Yaskawa INFORM job: X2_51(P)(-165,-90).JBI

/JOB
//NAME X2_51(P)(-165,-90)
//POS
///NPOS 337,337,337,21,0,0
///TOOL 0
///POSTYPE PULSE
///PULSE
C00000=39612,-76551,-106625,-19964,71626,-76894
C00001=136747,-74177,-105509,-19364,71994,-77223
C00002=161484,-91945,-110261,-14957,103238,-71453
C00003=160103,-106044,-63154,-4849,72775,-63697
C00004=161344,-104617,-58318,-4903,70612,-63188
C00005=161861,-103966,-56335,-4926,69759,-62977
C00006=161974,-102590,-54020,-4947,69050,-62909
C00007=162012,-102745,-54357,-4943,69180,-62902
C00008=163250,-104574,-55005,-4953,68713,-62462
C00009=162012,-102745,-54357,-4943,69180,-62902
C00010=160245,-104918,-61242,-4863,72187,-63625
C00011=171505,-139740,-90933,-7250,74874,-61360
C00012=160934,-120333,-86405,-7656,81002,-65284
C00013=161678,-120105,-82177,-7691,78608,-64883
C00014=162014,-119639,-79976,-7711,77534,-64702
C00015=162103,-118683,-78296,-7724,77005,-64638
C00016=162142,-118788,-78603,-7719,77142,-64634
C00017=163383,-121045,-79330,-7709,76552,-64175
C00018=162142,-118788,-78603,-7719,77142,-64634
C00019=161077,-119352,-84635,-7663,80435,-65200
C00020=170862,-154578,-108681,-8518,79424,-59558
C00021=160995,-130363,-103106,-9103,87223,-63446
C00022=161741,-131140,-99278,-9095,84585,-62999
C00023=162088,-130949,-97067,-9096,83376,-62793
C00024=162168,-130176,-95642,-9101,82912,-62732
C00025=162238,-130240,-95916,-9096,83053,-62718
C00026=163482,-133028,-96761,-9062,82290,-62238
C00027=162238,-130240,-95916,-9096,83053,-62718
C00028=161170,-129514,-101410,-9099,86642,-63344
C00029=164342,-146461,-115997,5708,80531,-78436
C00030=172620,-131260,-102348,10866,75066,-76115
C00031=174663,-130573,-98097,10735,72570,-75614
C00032=175557,-129771,-95630,10687,71364,-75403
C00033=175655,-129031,-94295,10701,70918,-75408
C00034=175682,-129209,-94620,10692,71020,-75389
C00035=177260,-131621,-95369,10541,70050,-74910
C00036=175682,-129209,-94620,10692,71020,-75389
C00037=172786,-130448,-100678,10875,74444,-76112
C00038=185712,-152871,-107287,9933,65474,-72285
C00039=172557,-120691,-85253,11157,70075,-76596
C00040=174600,-119310,-80674,11059,67728,-76082
C00041=175498,-118200,-77996,11031,66549,-75868
C00042=175592,-117418,-76647,11054,66116,-75875
C00043=175604,-117590,-76985,11043,66232,-75860
C00044=177181,-119548,-77634,10892,65428,-75363
C00045=175604,-117590,-76985,11043,66232,-75860
C00046=172709,-119718,-83491,11178,69480,-76597
C00047=183041,-134830,-88553,10500,63578,-73433
C00048=171873,-105200,-60293,14264,60373,-76350
C00049=174332,-102742,-55136,14143,58110,-75711
C00050=175369,-101410,-52567,14107,57068,-75452
C00051=175489,-100273,-50681,14176,56489,-75483
C00052=175484,-100515,-51075,14158,56604,-75470
C00053=177059,-102096,-51658,13960,55908,-74954
C00054=175484,-100515,-51075,14158,56604,-75470
C00055=174474,-101588,-53199,14210,57504,-75737
C00056=172007,-104102,-58400,14326,59768,-76379
C00057=145534,-132844,-96218,416,74991,-72838
C00058=145515,-153724,-122450,337,32933,-72823
C00059=145515,-153724,-122450,337,32933,-72823
C00060=145977,-137385,-98995,123,44015,-76512
C00061=126650,-119622,-94060,17558,35096,-87270
C00062=146093,-91262,-32695,-9242,9662,-72789
C00063=160671,-30783,15668,-32982,16065,-44517
C00064=161338,-23358,24708,-37738,14871,-42214
C00065=161591,-20267,28531,-39994,14370,-41134
C00066=161710,-18499,31905,-43322,13534,-39587
C00067=161697,-18674,31599,-43019,13601,-39728
C00068=160818,-16173,33693,-41566,13229,-40545
C00069=161697,-18674,31599,-43019,13601,-39728
C00070=161443,-21835,27676,-40467,14093,-40942
C00071=160779,-29405,18429,-35142,15276,-43501
C00072=135154,-32069,12634,-42029,20998,-54645
C00073=134732,-25138,21651,-45349,19348,-53134
C00074=134570,-22247,25451,-46978,18672,-52394
C00075=134606,-20594,28698,-49618,17908,-51149
C00076=134580,-20854,28257,-49268,17988,-51317
C00077=134270,-18078,30511,-48869,17866,-51557
C00078=134580,-20854,28257,-49268,17988,-51317
C00079=135167,-30880,15161,-43750,20301,-53823
C00080=130526,-37728,8761,-34606,19495,-58724
C00081=121050,-28931,19594,-23215,15148,-65580
C00082=121021,-21638,29205,-26791,13167,-63944
C00083=121010,-18566,33292,-28698,12330,-63076
C00084=121003,-15436,36219,-29112,12158,-62888
C00085=120965,-16234,35448,-28882,12203,-63000
C00086=120957,-14841,38575,-31824,11150,-61665
C00087=120965,-16234,35448,-28882,12203,-63000
C00088=121002,-26728,21497,-23181,15100,-65604
C00089=121044,-28941,19424,-23061,15238,-65652
C00090=121016,-21660,29021,-26586,13257,-64038
C00091=121005,-18594,33102,-28462,12419,-63184
C00092=120998,-15466,36026,-28869,12247,-63000
C00093=120970,-16325,35175,-28625,12311,-63116
C00094=120961,-14943,38290,-31508,11257,-61807
C00095=120970,-16325,35175,-28625,12311,-63116
C00096=121007,-26794,21256,-23025,15206,-65675
C00097=146102,-87320,-26882,-11020,8134,-71987
C00098=145977,-137385,-98995,123,44015,-76512
C00099=112492,-157991,-119063,-2457,0,-76621
C00100=-11604,-169116,-125244,-11553,23484,-75880
C00101=-142186,-149365,-128787,911,0,-68169
C00102=-169394,-149435,-128797,930,71008,-68172
C00103=-146318,-131671,-100763,953,62874,-68185
C00104=-112829,-124197,-91749,2815,37541,-68231
C00105=-106317,-89557,-31431,-13456,10069,-57380
C00106=-82305,-48194,-2702,-1068,13384,-54980
C00107=-80735,-41443,4673,-5524,12373,-52723
C00108=-80143,-38689,7738,-7432,11949,-51767
C00109=-80007,-37233,10634,-8542,10936,-51243
C00110=-79998,-37162,10484,-8474,11064,-51273
C00111=-80961,-34830,12178,-5427,11144,-52800
C00112=-79998,-37162,10484,-8474,11064,-51273
C00113=-80428,-35938,10350,-6726,11733,-52131
C00114=-78778,-34690,11115,-11291,12069,-49811
C00115=-80428,-35938,10350,-6726,11733,-52131
C00116=-82562,-45500,-282,-411,13276,-55316
C00117=-92230,-47187,-3616,-43240,24199,-57639
C00118=-93096,-40890,4303,-45146,22607,-56839
C00119=-93429,-38304,7591,-46074,21957,-56442
C00120=-93338,-36887,10462,-48076,21279,-55468
C00121=-93324,-37096,10094,-47861,21367,-55569
C00122=-93984,-34586,11898,-46952,21176,-56108
C00123=-93324,-37096,10094,-47861,21367,-55569
C00124=-92116,-46106,-1290,-44710,23611,-56904
C00125=-91073,-53322,-8580,-41986,25230,-57812
C00126=-91939,-47488,-3032,-40883,24993,-58457
C00127=-92774,-41247,4932,-42701,23345,-57694
C00128=-93096,-38682,8241,-43585,22671,-57316
C00129=-93741,-35973,10491,-43009,22389,-57697
C00130=-93557,-36801,9788,-43160,22476,-57594
C00131=-93351,-35803,12350,-45165,21793,-56596
C00132=-93557,-36801,9788,-43160,22476,-57594
C00133=-92437,-45645,-1602,-40370,24830,-58783
C00134=-106116,-47899,-3414,-24973,19848,-68149
C00135=-106551,-41527,4610,-26418,18218,-67531
C00136=-106718,-38911,7943,-27146,17534,-67215
C00137=-107051,-36097,10252,-26581,17460,-67530
C00138=-106917,-36892,9642,-26842,17469,-67388
C00139=-106813,-35930,12180,-28635,16550,-66536
C00140=-106917,-36892,9642,-26842,17469,-67388
C00141=-106334,-45915,-1841,-24600,19835,-68356
C00142=-112836,-101934,-56773,3722,27473,-393
C00143=-146326,-133616,-103789,948,63737,26
C00144=-169394,-149435,-128797,930,71008,40
C00145=-130640,-113336,-116882,-25805,15754,2900
C00146=-135014,-119633,-103449,-15272,86576,5177
C00147=-145520,-105980,-62980,746,70150,73322
C00148=-146362,-104694,-58180,786,67864,73018
C00149=-146742,-103661,-55476,805,66734,72879
C00150=-146802,-102720,-53893,810,66245,72855
C00151=-146820,-102923,-54246,810,66358,72850
C00152=-147635,-104920,-54937,842,65765,72565
C00153=-146820,-102923,-54246,810,66358,72850
C00154=-145619,-104907,-61084,752,69535,73285
C00155=-171454,-106797,-63241,1567,70253,64421
C00156=-173073,-105087,-58310,1635,68130,63837
C00157=-173822,-103661,-55199,1669,66963,63564
C00158=-173907,-102906,-53963,1677,66592,63529
C00159=-173899,-103121,-54319,1675,66700,63533
C00160=-175454,-104758,-54906,1725,66251,62992
C00161=-173899,-103121,-54319,1675,66700,63533
C00162=-171598,-105684,-61333,1577,69654,64364
C00163=-171851,-142113,-91727,1629,69899,64268
C00164=-158429,-121713,-86926,1143,76935,68953
C00165=-159677,-121086,-82564,1192,74590,68504
C00166=-160262,-120091,-79675,1217,73333,68291
C00167=-160325,-119479,-78625,1221,73002,68266
C00168=-160351,-119548,-78930,1221,73155,68259
C00169=-161558,-121835,-79657,1263,72445,67838
C00170=-160351,-119548,-78930,1221,73155,68259
C00171=-158575,-120647,-85141,1149,76386,68898
C00172=-146231,-120412,-85894,9154,79904,67922
C00173=-146532,-120200,-81655,9220,77469,67638
C00174=-146707,-119317,-78712,9263,76149,67479
C00175=-146746,-118772,-77764,9274,75853,67443
C00176=-146790,-118881,-78072,9269,75989,67438
C00177=-147605,-121338,-78846,9287,75305,67107
C00178=-146790,-118881,-78072,9269,75989,67438
C00179=-146355,-119421,-84118,9167,79342,67838
C00180=-155393,-157537,-108482,12071,78573,60028
C00181=-146205,-130572,-102237,12226,86761,64000
C00182=-146506,-131303,-98376,12244,84115,63635
C00183=-146668,-130963,-95920,12261,82832,63453
C00184=-146721,-130297,-94717,12268,82450,63397
C00185=-146765,-130382,-95017,12263,82595,63396
C00186=-147581,-133401,-95913,12252,81739,63030
C00187=-146765,-130382,-95017,12263,82595,63396
C00188=-146330,-129706,-100552,12225,86202,63901
C00189=-158435,-132386,-103934,1126,81916,68996
C00190=-159685,-132645,-99938,1172,79342,68546
C00191=-160276,-131966,-97169,1195,77996,68332
C00192=-160335,-131435,-96228,1198,77691,68309
C00193=-160363,-131651,-96568,1198,77790,68300
C00194=-161574,-134495,-97414,1239,76868,67878
C00195=-160363,-131651,-96568,1198,77790,68300
C00196=-158581,-131628,-102288,1132,81296,68941
C00197=-156763,-87672,-103760,774,105674,87516
C00198=-169394,-149435,-128797,930,71008,83169
C00199=-150414,-86289,-54081,-474,90119,72869
C00200=-151266,-87748,-50943,-622,87433,72599
C00201=-152488,-87428,-48859,-834,86309,72204
C00202=-148147,-89589,-49139,4425,86731,74395
C00203=-146818,-89870,-51113,4706,87732,74872
C00204=-146666,-88304,-54215,4739,90428,75023
C00205=-138939,-90669,-55596,-9574,86239,77137
C00206=-140404,-91758,-52256,-9806,83488,76860
C00207=-142815,-91310,-50219,-10159,82191,76162
C00208=-154710,-86462,-48344,-11637,81955,72207
C00209=-152664,-87123,-50558,-11375,83242,72777
C00210=-150783,-86165,-53887,-11117,85991,73164
C00211=-154131,-121950,-82387,-8712,85987,67425
C00212=-148025,-100109,-75076,-5665,93909,72754
C00213=-148831,-100312,-70826,-5762,91146,72606
C00214=-146468,-101528,-70218,-8213,89409,73952
C00215=-156895,-95901,-68057,-9567,89811,70382
C00216=-156895,-97491,-71326,-9574,90990,70292
C00217=-153017,-102427,-75547,-11357,90518,71992
C00218=-151529,-98458,-73502,4508,98276,66494
C00219=-151321,-97538,-69606,4526,96344,66497
C00220=-152185,-98274,-68237,4332,95173,66163
C00221=-146393,-100560,-68313,8882,94911,67867
C00222=-146800,-100443,-69693,10119,95679,69043
C00223=-151558,-100768,-73356,9121,98301,67607
C00224=-156292,-129361,-96058,9643,101176,59304
C00225=-152402,-99580,-86113,11137,109464,61436
C00226=-153129,-103579,-84123,10707,106340,60878
C00227=-153762,-104985,-82590,10439,104784,60514
C00228=-145239,-109230,-83490,14196,102512,63288
C00229=-141027,-109993,-86316,13674,102607,64868
C00230=-140829,-106100,-88459,13958,105801,65311
C00231=-138968,-107947,-91550,-9748,99253,76121
C00232=-140436,-111637,-89327,-9854,95856,75879
C00233=-143265,-112181,-87516,-10198,94133,75040
C00234=-154691,-105452,-85498,-11618,94761,71024
C00235=-152715,-105048,-87091,-11430,96209,71575
C00236=-150832,-103395,-97227,-11518,103428,71561
C00237=-124659,-112995,-107713,-28856,68615,65766
C00238=-126218,-114256,-117174,-36511,17097,46518
C00239=-148561,-148351,-134746,-2636,59820,4885
C00240=-157191,-155093,-133027,-2423,70817,-63833
C00241=-146254,-116377,-77147,999,56200,-68180
C00242=-107275,-71407,-14739,-39799,20998,-48318
C00243=-107236,-64792,-7336,-41859,20126,-47330
C00244=-107209,-61980,-4011,-43007,19687,-46782
C00245=-70112,-45989,3773,-54150,40066,-34286
C00246=-69774,-48485,443,-53474,40707,-34620
C00247=-68604,-54637,-7231,-52245,42284,-35133
C00248=-92320,-90311,-38101,-17507,21359,-69759
C00249=-104434,-95533,-39177,3441,13241,-85394
C00250=-104568,-88850,-32673,3945,12680,-85644
C00251=-104520,-86387,-29909,3952,12244,-85640
C00252=-67588,-70566,-24092,-47976,27768,-56046
C00253=-72044,-71463,-22366,-44090,19939,-45466
C00254=-72907,-74424,-25211,-42700,19719,-46246
C00255=-73002,-81137,-31884,-41377,20172,-46887
C00256=-111917,-134748,-95138,2307,25782,-38985
C00257=-112830,-118606,-82850,2996,34941,-68234
C00258=-146284,-125214,-92772,982,57715,-68183
C00259=-169394,-149435,-128797,930,71008,-68172
C00260=-133816,-149354,-128786,835,13880,-68173
C00261=-90671,-157974,-126979,-5410,0,-71957
C00262=-11604,-169116,-125244,-11553,23484,-75880
C00263=137287,-84892,-120500,-10191,64594,-76446
C00264=160620,-101266,-113002,-23179,68693,-67515
C00265=177556,-94372,-53425,-385,88988,-62741
C00266=179326,-95097,-49878,3,86437,-62164
C00267=179814,-95288,-47635,109,84959,-62011
C00268=167774,-103484,-50203,-2536,82158,-65798
C00269=167400,-103593,-52544,-2612,83531,-65942
C00270=166065,-103008,-56268,-2894,86078,-66424
C00271=166312,-127479,-80936,-5864,94766,-53062
C00272=158392,-93304,-69893,-8747,104686,-56339
C00273=159554,-95674,-67229,-8288,101981,-55739
C00274=159445,-96667,-65849,-8272,100624,-55685
C00275=147725,-102887,-67985,-11495,97353,-59463
C00276=147678,-102382,-69650,-11553,98605,-59595
C00277=146987,-100069,-72442,-11867,101354,-60101
C00278=154304,-136297,-99225,-6964,97533,-61473
C00279=152227,-100568,-87835,-8146,108504,-62877
C00280=153116,-104646,-85864,-7761,105315,-62341
C00281=159148,-124823,-92360,-9877,92486,-59205
C00282=144137,-132852,-94532,-12005,87729,-63907
C00283=143944,-126885,-94638,-11486,92524,-64465
C00284=145540,-135687,-103511,-12475,90096,-63617
C00285=148082,-100818,-99733,10674,107205,-74531
C00286=152803,-93035,-83606,23107,96838,-80328
C00287=154879,-96218,-81430,23079,93509,-80208
C00288=162734,-110375,-86778,19923,82294,-79319
C00289=172936,-99666,-82887,19315,82782,-75563
C00290=164774,-87312,-77814,23533,92874,-76681
C00291=167890,-98830,-87724,19097,86606,-76775
C00292=158633,-112297,-90822,23483,90242,-79469
C00293=153117,-105481,-75293,18446,87539,-80566
C00294=154070,-103992,-71187,18555,85650,-80517
C00295=161541,-113229,-74370,16909,77144,-78922
C00296=171872,-105466,-71629,16874,77244,-75258
C00297=165515,-96039,-68345,19422,85228,-76531
C00298=163213,-94486,-71315,19256,88254,-76871
C00299=168945,-117983,-78283,23930,79136,-80745
C00300=162859,-103904,-55417,26052,71934,-81289
C00301=166467,-103150,-51264,26590,68911,-80665
C00302=174261,-106144,-51758,25332,63333,-78665
C00303=185047,-97716,-49331,24449,62895,-74631
C00304=178605,-94860,-48677,26497,67666,-76392
C00305=170055,-106805,-62873,25975,72582,-78466
C00306=152982,-88821,-92221,4904,67346,-32106
C00307=145515,-153724,-122450,337,32933,46
C00308=145515,-153724,-122450,337,32933,46
C00309=145977,-137385,-98995,123,44015,44
C00310=84186,-58858,-9027,66870,52124,39353
C00311=87105,-53815,-2337,68349,49752,38990
C00312=88013,-52041,490,69129,48884,38670
C00313=128614,-57932,-1955,73297,23821,44535
C00314=127846,-60584,-5316,71867,24516,45096
C00315=125900,-66978,-12435,69921,26079,45715
C00316=123713,-86623,-29625,34014,27338,1409
C00317=121149,-57675,-2785,-2636,26737,-48399
C00318=121132,-57328,-2241,-2634,26580,-48403
C00319=121104,-54911,-3160,-2183,31831,-48629
C00320=158495,-44767,2170,-23903,39526,-29988
C00321=121132,-57338,-2123,-2642,26502,-48399
C00322=121149,-57624,-2567,-2646,26629,-48394
C00323=145977,-137385,-98995,123,44015,44
C00324=141323,-155575,-119470,2858,47354,-2051
C00325=136193,-54528,-31246,1392,38939,57192
C00326=133673,-4879,12102,671,34805,86301
C00327=129645,-10071,18191,6510,19037,82612
C00328=146465,2091,28934,7064,17500,85725
C00329=143182,-12622,11657,11660,20903,83241
C00330=129180,-33068,-6989,1774,26259,77639
C00331=129999,-18466,14492,894,20530,78149
C00332=103012,-15842,16412,36484,27005,57754
C00333=109108,-49067,-22735,24370,30989,64550
C00334=115971,-133718,-81561,22438,22383,66198
C00335=115971,-174253,-123740,18555,27203,68106
C00336=39612,-76551,-106625,-19964,71626,-76894
BC00000=295309,515546,1075139
BC00001=353519,294132,1075139
BC00002=353519,214242,1075139
BC00003=331202,150916,1075139
BC00004=331202,150916,1075139
BC00005=331202,150916,1075139
BC00006=331202,150916,1075139
BC00007=331202,150916,1075139
BC00008=331202,150916,1075139
BC00009=331202,150916,1075139
BC00010=331202,150916,1075139
BC00011=324436,118777,1075139
BC00012=324436,118777,1075139
BC00013=324436,118777,1075139
BC00014=324436,118777,1075139
BC00015=324436,118777,1075139
BC00016=324436,118777,1075139
BC00017=324436,118777,1075139
BC00018=324436,118777,1075139
BC00019=324436,118777,1075139
BC00020=321391,89351,1075139
BC00021=321391,89351,1075139
BC00022=321391,89351,1075139
BC00023=321391,89351,1075139
BC00024=321391,89351,1075139
BC00025=321391,89351,1075139
BC00026=321391,89351,1075139
BC00027=321391,89351,1075139
BC00028=321391,89351,1075139
BC00029=308521,79020,1075139
BC00030=308521,79020,1075139
BC00031=308521,79020,1075139
BC00032=308521,79020,1075139
BC00033=308521,79020,1075139
BC00034=308521,79020,1075139
BC00035=308521,79020,1075139
BC00036=308521,79020,1075139
BC00037=308521,79020,1075139
BC00038=308521,79020,1075139
BC00039=308654,108079,1075139
BC00040=308654,108079,1075139
BC00041=308654,108079,1075139
BC00042=308654,108079,1075139
BC00043=308654,108079,1075139
BC00044=308654,108079,1075139
BC00045=308654,108079,1075139
BC00046=308654,108079,1075139
BC00047=308654,108079,1075139
BC00048=315387,142542,1075139
BC00049=315387,142542,1075139
BC00050=315387,142542,1075139
BC00051=315387,142542,1075139
BC00052=315387,142542,1075139
BC00053=315387,142542,1075139
BC00054=315387,142542,1075139
BC00055=315387,142542,1075139
BC00056=315387,142542,1075139
BC00057=334019,183746,1075139
BC00058=334019,229146,1075139
BC00059=369517,393170,1075139
BC00060=369517,393170,1075139
BC00061=309272,310148,725948
BC00062=299317,286166,1016538
BC00063=320949,304869,1075139
BC00064=320949,304869,1075139
BC00065=320949,304869,1075139
BC00066=320949,304869,1075139
BC00067=320949,304869,1075139
BC00068=320949,304869,1075139
BC00069=320949,304869,1075139
BC00070=320949,304869,1075139
BC00071=320949,304869,1075139
BC00072=287778,324241,1075139
BC00073=287778,324241,1075139
BC00074=287778,324241,1075139
BC00075=287778,324241,1075139
BC00076=287778,324241,1075139
BC00077=287778,324241,1075139
BC00078=287778,324241,1075139
BC00079=287778,324241,1075139
BC00080=279976,328662,1075139
BC00081=264373,337505,1075139
BC00082=264373,337505,1075139
BC00083=264373,337505,1075139
BC00084=264373,337505,1075139
BC00085=264373,337505,1075139
BC00086=264373,337505,1075139
BC00087=264373,337505,1075139
BC00088=264373,337505,1075139
BC00089=317151,337442,1075139
BC00090=317151,337442,1075139
BC00091=317151,337442,1075139
BC00092=317151,337442,1075139
BC00093=317151,337442,1075139
BC00094=317151,337442,1075139
BC00095=317151,337442,1075139
BC00096=317151,337442,1075139
BC00097=324891,309494,1043787
BC00098=369517,393170,1075139
BC00099=372480,297840,1075139
BC00100=335939,159824,1075139
BC00101=387142,-83097,1073718
BC00102=387142,-83097,1073718
BC00103=354260,-55239,919482
BC00104=302473,-54215,830727
BC00105=299756,-34503,1018031
BC00106=266432,-33337,1015863
BC00107=266432,-33337,1015863
BC00108=266432,-33337,1015863
BC00109=266432,-33337,1015863
BC00110=266432,-33337,1015863
BC00111=266432,-33337,1015863
BC00112=266432,-33337,1015863
BC00113=266432,-33337,1015863
BC00114=266432,-33337,1015863
BC00115=266432,-33337,1015863
BC00116=266432,-33337,1015863
BC00117=284169,-51063,1035355
BC00118=284169,-51063,1035355
BC00119=284169,-51063,1035355
BC00120=284169,-51063,1035355
BC00121=284169,-51063,1035355
BC00122=284169,-51063,1035355
BC00123=284169,-51063,1035355
BC00124=284169,-51063,1035355
BC00125=283205,-57233,1023653
BC00126=282402,-62375,1013902
BC00127=282402,-62375,1013902
BC00128=282402,-62375,1013902
BC00129=282402,-62375,1013902
BC00130=282402,-62375,1013902
BC00131=282402,-62375,1013902
BC00132=282402,-62375,1013902
BC00133=282402,-62375,1013902
BC00134=251376,-67725,1013804
BC00135=251376,-67725,1013804
BC00136=251376,-67725,1013804
BC00137=251376,-67725,1013804
BC00138=251376,-67725,1013804
BC00139=251376,-67725,1013804
BC00140=251376,-67725,1013804
BC00141=251376,-67725,1013804
BC00142=302473,-54215,999708
BC00143=354260,-55239,903923
BC00144=387142,-83097,1073718
BC00145=343892,52052,1075139
BC00146=340737,74809,1075139
BC00147=324434,99527,1075139
BC00148=324434,99527,1075139
BC00149=324434,99527,1075139
BC00150=324434,99527,1075139
BC00151=324434,99527,1075139
BC00152=324434,99527,1075139
BC00153=324434,99527,1075139
BC00154=324434,99527,1075139
BC00155=316013,112625,1075139
BC00156=316013,112625,1075139
BC00157=316013,112625,1075139
BC00158=316013,112625,1075139
BC00159=316013,112625,1075139
BC00160=316013,112625,1075139
BC00161=316013,112625,1075139
BC00162=316013,112625,1075139
BC00163=304877,137904,1075139
BC00164=304877,137904,1075139
BC00165=304877,137904,1075139
BC00166=304877,137904,1075139
BC00167=304877,137904,1075139
BC00168=304877,137904,1075139
BC00169=304877,137904,1075139
BC00170=304877,137904,1075139
BC00171=304877,137904,1075139
BC00172=308833,132707,1075139
BC00173=308833,132707,1075139
BC00174=308833,132707,1075139
BC00175=308833,132707,1075139
BC00176=308833,132707,1075139
BC00177=308833,132707,1075139
BC00178=308833,132707,1075139
BC00179=308833,132707,1075139
BC00180=303080,163439,1075139
BC00181=303080,163439,1075139
BC00182=303080,163439,1075139
BC00183=303080,163439,1075139
BC00184=303080,163439,1075139
BC00185=303080,163439,1075139
BC00186=303080,163439,1075139
BC00187=303080,163439,1075139
BC00188=303080,163439,1075139
BC00189=304913,167110,1075139
BC00190=304913,167110,1075139
BC00191=304913,167110,1075139
BC00192=304913,167110,1075139
BC00193=304913,167110,1075139
BC00194=304913,167110,1075139
BC00195=304913,167110,1075139
BC00196=304913,167110,1075139
BC00197=340038,100851,1073718
BC00198=340038,100851,1073718
BC00199=318440,111564,1057595
BC00200=318440,111564,1057595
BC00201=318440,111564,1057593
BC00202=318440,111564,1057595
BC00203=318440,111564,1057595
BC00204=318440,111564,1057595
BC00205=310795,111718,1057781
BC00206=310795,111718,1057781
BC00207=310795,111718,1057781
BC00208=310795,111718,1057781
BC00209=310795,111718,1057781
BC00210=310795,111718,1057781
BC00211=314493,146927,1075139
BC00212=311302,144606,1075139
BC00213=311302,144606,1075139
BC00214=311090,144452,1075139
BC00215=311090,144452,1075139
BC00216=311090,144452,1075139
BC00217=310912,144322,1075139
BC00218=309663,144665,1075139
BC00219=309663,144665,1075139
BC00220=309663,144665,1075139
BC00221=309663,144665,1075139
BC00222=309663,144665,1075139
BC00223=309663,144665,1075139
BC00224=293187,178635,1075139
BC00225=300015,175953,1075139
BC00226=300015,175953,1075139
BC00227=300015,175953,1075139
BC00228=300015,175953,1075139
BC00229=300015,175953,1075139
BC00230=300015,175953,1075139
BC00231=311011,173433,1075139
BC00232=311011,173433,1075139
BC00233=311011,173433,1075139
BC00234=311011,173433,1075139
BC00235=311011,173433,1075139
BC00236=311011,173433,1075139
BC00237=311721,119711,1075139
BC00238=312616,52052,1075139
BC00239=363630,-40460,1074166
BC00240=387142,-83097,1073718
BC00241=354260,-55239,1037445
BC00242=264595,-32771,1007498
BC00243=264595,-32771,1007498
BC00244=264595,-32771,1007498
BC00245=264595,-32771,1007498
BC00246=264595,-32771,1007498
BC00247=264595,-32771,1007498
BC00248=281388,-13085,953726
BC00249=292015,-7655,938135
BC00250=292015,-7655,938135
BC00251=292015,-7655,938135
BC00252=292015,-7655,938135
BC00253=292015,-7655,938135
BC00254=292015,-7655,938135
BC00255=292015,-7655,938135
BC00256=305209,-34503,728557
BC00257=302473,-54215,875335
BC00258=354260,-55239,995141
BC00259=387142,-83097,1073718
BC00260=387142,-83097,1073718
BC00261=392686,38993,1074432
BC00262=335939,159824,1075139
BC00263=353801,266119,1075139
BC00264=381880,223521,1075139
BC00265=325796,119524,1075139
BC00266=325796,119524,1075139
BC00267=325796,119524,1075139
BC00268=325796,119524,1075139
BC00269=325796,119524,1075139
BC00270=325796,119524,1075139
BC00271=298605,97380,1075139
BC00272=306786,105313,1075139
BC00273=306786,105313,1075139
BC00274=306786,105313,1075139
BC00275=306786,105313,1075139
BC00276=306786,105313,1075139
BC00277=306786,105313,1075139
BC00278=296424,73357,1075139
BC00279=304436,81384,1075139
BC00280=304436,81384,1075139
BC00281=304436,81384,1075139
BC00282=304436,81384,1075139
BC00283=304436,81384,1075139
BC00284=304436,81384,1075139
BC00285=314150,82141,1075139
BC00286=318449,85788,1075139
BC00287=318449,85788,1075139
BC00288=318449,85788,1075139
BC00289=318449,85788,1075139
BC00290=318449,85788,1075139
BC00291=318449,85788,1075139
BC00292=319675,83840,1075139
BC00293=303619,103646,1075139
BC00294=303619,103646,1075139
BC00295=303619,103646,1075139
BC00296=303619,103646,1075139
BC00297=303619,103646,1075139
BC00298=303619,103646,1075139
BC00299=318801,93459,1075139
BC00300=319660,117178,1064998
BC00301=319660,117178,1064998
BC00302=319660,117178,1064998
BC00303=319660,117178,1064998
BC00304=319660,117178,1064998
BC00305=319660,117178,1064998
BC00306=339598,204159,1070920
BC00307=334019,229146,1075139
BC00308=369517,393170,1075139
BC00309=369517,393170,1075139
BC00310=279240,278181,995341
BC00311=279240,278181,995341
BC00312=279240,278181,995341
BC00313=279240,278181,995341
BC00314=279240,278181,995341
BC00315=279240,278181,995341
BC00316=306644,283045,1033505
BC00317=336539,288351,1075139
BC00318=333822,285094,1054529
BC00319=332736,283791,1045508
BC00320=332727,283791,1045508
BC00321=279880,285191,1054163
BC00322=282597,288448,1075139
BC00323=369517,393170,1075139
BC00324=209346,479306,1075139
BC00325=169680,397657,995179
BC00326=150190,357539,955892
BC00327=150190,357539,955892
BC00328=150190,357539,955892
BC00329=150190,357539,955892
BC00330=150190,357539,955892
BC00331=150190,357539,955892
BC00332=150190,357539,955892
BC00333=150190,357539,955892
BC00334=150190,357539,955892
BC00335=150190,552519,961001
BC00336=295309,515546,1075139
EC00000=1463287,372643
EC00001=1463287,372643
EC00002=1463287,372643
EC00003=1463287,372643
EC00004=1463287,372643
EC00005=1463287,372643
EC00006=1463287,372643
EC00007=1463287,372643
EC00008=1463287,372643
EC00009=1463287,372643
EC00010=1463287,372643
EC00011=1463287,372643
EC00012=1463287,372643
EC00013=1463287,372643
EC00014=1463287,372643
EC00015=1463287,372643
EC00016=1463287,372643
EC00017=1463287,372643
EC00018=1463287,372643
EC00019=1463287,372643
EC00020=1463287,372643
EC00021=1463287,372643
EC00022=1463287,372643
EC00023=1463287,372643
EC00024=1463287,372643
EC00025=1463287,372643
EC00026=1463287,372643
EC00027=1463287,372643
EC00028=1463287,372643
EC00029=1463287,372643
EC00030=1463287,372643
EC00031=1463287,372643
EC00032=1463287,372643
EC00033=1463287,372643
EC00034=1463287,372643
EC00035=1463287,372643
EC00036=1463287,372643
EC00037=1463287,372643
EC00038=1463287,372643
EC00039=1463287,372643
EC00040=1463287,372643
EC00041=1463287,372643
EC00042=1463287,372643
EC00043=1463287,372643
EC00044=1463287,372643
EC00045=1463287,372643
EC00046=1463287,372643
EC00047=1463287,372643
EC00048=1463287,372643
EC00049=1463287,372643
EC00050=1463287,372643
EC00051=1463287,372643
EC00052=1463287,372643
EC00053=1463287,372643
EC00054=1463287,372643
EC00055=1463287,372643
EC00056=1463287,372643
EC00057=1463287,372643
EC00058=1463287,372643
EC00059=1463287,372643
EC00060=1463287,372643
EC00061=1463287,372643
EC00062=1463287,372643
EC00063=1463287,372643
EC00064=1463287,372643
EC00065=1463287,372643
EC00066=1463287,372643
EC00067=1463287,372643
EC00068=1463287,372643
EC00069=1463287,372643
EC00070=1463287,372643
EC00071=1463287,372643
EC00072=1463287,372643
EC00073=1463287,372643
EC00074=1463287,372643
EC00075=1463287,372643
EC00076=1463287,372643
EC00077=1463287,372643
EC00078=1463287,372643
EC00079=1463287,372643
EC00080=1463287,372643
EC00081=1463287,372643
EC00082=1463287,372643
EC00083=1463287,372643
EC00084=1463287,372643
EC00085=1463287,372643
EC00086=1463287,372643
EC00087=1463287,372643
EC00088=1463287,372643
EC00089=1463287,372643
EC00090=1463287,372643
EC00091=1463287,372643
EC00092=1463287,372643
EC00093=1463287,372643
EC00094=1463287,372643
EC00095=1463287,372643
EC00096=1463287,372643
EC00097=1463287,372643
EC00098=1463287,372643
EC00099=1463287,372643
EC00100=1595090,-179995
EC00101=1729339,-740307
EC00102=1729339,-740307
EC00103=1729339,-740307
EC00104=1729339,-740307
EC00105=1729339,-740307
EC00106=1729339,-740307
EC00107=1729339,-740307
EC00108=1729339,-740307
EC00109=1729339,-740307
EC00110=1729339,-740307
EC00111=1729339,-740307
EC00112=1729339,-740307
EC00113=1729339,-740307
EC00114=1729339,-740307
EC00115=1729339,-740307
EC00116=1729339,-740307
EC00117=1729339,-740307
EC00118=1729339,-740307
EC00119=1729339,-740307
EC00120=1729339,-740307
EC00121=1729339,-740307
EC00122=1729339,-740307
EC00123=1729339,-740307
EC00124=1729339,-740307
EC00125=1729339,-740307
EC00126=1729339,-740307
EC00127=1729339,-740307
EC00128=1729339,-740307
EC00129=1729339,-740307
EC00130=1729339,-740307
EC00131=1729339,-740307
EC00132=1729339,-740307
EC00133=1729339,-740307
EC00134=1729339,-740307
EC00135=1729339,-740307
EC00136=1729339,-740307
EC00137=1729339,-740307
EC00138=1729339,-740307
EC00139=1729339,-740307
EC00140=1729339,-740307
EC00141=1729339,-740307
EC00142=1729339,-740307
EC00143=1729339,-740307
EC00144=1729339,-740307
EC00145=1729339,-740307
EC00146=1729339,-740307
EC00147=1729339,-740307
EC00148=1729339,-740307
EC00149=1729339,-740307
EC00150=1729339,-740307
EC00151=1729339,-740307
EC00152=1729339,-740307
EC00153=1729339,-740307
EC00154=1729339,-740307
EC00155=1729339,-740307
EC00156=1729339,-740307
EC00157=1729339,-740307
EC00158=1729339,-740307
EC00159=1729339,-740307
EC00160=1729339,-740307
EC00161=1729339,-740307
EC00162=1729339,-740307
EC00163=1729339,-740307
EC00164=1729339,-740307
EC00165=1729339,-740307
EC00166=1729339,-740307
EC00167=1729339,-740307
EC00168=1729339,-740307
EC00169=1729339,-740307
EC00170=1729339,-740307
EC00171=1729339,-740307
EC00172=1729339,-740307
EC00173=1729339,-740307
EC00174=1729339,-740307
EC00175=1729339,-740307
EC00176=1729339,-740307
EC00177=1729339,-740307
EC00178=1729339,-740307
EC00179=1729339,-740307
EC00180=1729339,-740307
EC00181=1729339,-740307
EC00182=1729339,-740307
EC00183=1729339,-740307
EC00184=1729339,-740307
EC00185=1729339,-740307
EC00186=1729339,-740307
EC00187=1729339,-740307
EC00188=1729339,-740307
EC00189=1729339,-740307
EC00190=1729339,-740307
EC00191=1729339,-740307
EC00192=1729339,-740307
EC00193=1729339,-740307
EC00194=1729339,-740307
EC00195=1729339,-740307
EC00196=1729339,-740307
EC00197=1729339,-740307
EC00198=1729339,-740307
EC00199=1729339,-740307
EC00200=1729339,-740307
EC00201=1729340,-740306
EC00202=1729339,-740307
EC00203=1729339,-740307
EC00204=1729339,-740307
EC00205=1729339,-740307
EC00206=1729339,-740307
EC00207=1729339,-740307
EC00208=1729339,-740307
EC00209=1729339,-740307
EC00210=1729339,-740307
EC00211=1729339,-740307
EC00212=1729339,-740307
EC00213=1729339,-740307
EC00214=1729339,-740307
EC00215=1729339,-740307
EC00216=1729339,-740307
EC00217=1729339,-740307
EC00218=1729339,-740307
EC00219=1729339,-740307
EC00220=1729339,-740307
EC00221=1729339,-740307
EC00222=1729339,-740307
EC00223=1729339,-740307
EC00224=1729339,-740307
EC00225=1729339,-740307
EC00226=1729339,-740307
EC00227=1729339,-740307
EC00228=1729339,-740307
EC00229=1729339,-740307
EC00230=1729339,-740307
EC00231=1729339,-740307
EC00232=1729339,-740307
EC00233=1729339,-740307
EC00234=1729339,-740307
EC00235=1729339,-740307
EC00236=1729339,-740307
EC00237=1729339,-740307
EC00238=1729339,-740307
EC00239=1729339,-740307
EC00240=1729339,-740307
EC00241=1729339,-740307
EC00242=1729339,-740307
EC00243=1729339,-740307
EC00244=1729339,-740307
EC00245=1729339,-740307
EC00246=1729339,-740307
EC00247=1729339,-740307
EC00248=1729339,-740307
EC00249=1729339,-740307
EC00250=1729339,-740307
EC00251=1729339,-740307
EC00252=1729339,-740307
EC00253=1729339,-740307
EC00254=1729339,-740307
EC00255=1729339,-740307
EC00256=1729339,-740307
EC00257=1729339,-740307
EC00258=1729339,-740307
EC00259=1729339,-740307
EC00260=1729339,-740307
EC00261=1661867,-458699
EC00262=1595090,-179995
EC00263=1463287,372643
EC00264=1463287,372643
EC00265=1463287,372643
EC00266=1463287,372643
EC00267=1463287,372643
EC00268=1463287,372643
EC00269=1463287,372643
EC00270=1463287,372643
EC00271=1463287,372643
EC00272=1463287,372643
EC00273=1463287,372643
EC00274=1463287,372643
EC00275=1463287,372643
EC00276=1463287,372643
EC00277=1463287,372643
EC00278=1463287,372643
EC00279=1463287,372643
EC00280=1463287,372643
EC00281=1463287,372643
EC00282=1463287,372643
EC00283=1463287,372643
EC00284=1463287,372643
EC00285=1463287,372643
EC00286=1463287,372643
EC00287=1463287,372643
EC00288=1463287,372643
EC00289=1463287,372643
EC00290=1463287,372643
EC00291=1463287,372643
EC00292=1463287,372643
EC00293=1463287,372643
EC00294=1463287,372643
EC00295=1463287,372643
EC00296=1463287,372643
EC00297=1463287,372643
EC00298=1463287,372643
EC00299=1463287,372643
EC00300=1463287,372643
EC00301=1463287,372643
EC00302=1463287,372643
EC00303=1463287,372643
EC00304=1463287,372643
EC00305=1463287,372643
EC00306=1463287,372643
EC00307=1463287,372643
EC00308=1463287,372643
EC00309=1463287,372643
EC00310=1463287,372643
EC00311=1463287,372643
EC00312=1463287,372643
EC00313=1463287,372643
EC00314=1463287,372643
EC00315=1463287,372643
EC00316=1463287,372643
EC00317=1463287,372643
EC00318=1463287,372643
EC00319=1463287,372643
EC00320=1463287,372643
EC00321=1463287,372643
EC00322=1463287,372643
EC00323=1463287,372643
EC00324=1463287,372643
EC00325=1463287,372643
EC00326=1463287,372643
EC00327=1463287,372643
EC00328=1463287,372643
EC00329=1463287,372643
EC00330=1463287,372643
EC00331=1463287,372643
EC00332=1463287,372643
EC00333=1463287,372643
EC00334=1463287,372643
EC00335=1463287,372643
EC00336=1463287,372643
///POSTYPE BASE
///RECTAN
///RCONF 0,0,0,0,1,0,0,0,0,0,0,0,0,0,0,0,0,0,0,0,0,0,0,0
P00006=2.006,1.622,-0.565,0.0000,0.0000,0.0000
P00021=0.073,2.058,-0.109,0.0000,0.0000,0.0000
P00022=2.006,1.622,-0.565,0.0000,0.0000,0.0000
///RCONF 0,0,0,0,0,0,0,0,0,0,0,0,0,0,0,0,0,0,0,0,0,0,0,0
P00023=-2.957,-4.083,2.762,0.0000,0.0000,0.0000
P00024=-1.466,-0.226,-0.419,0.0000,0.0000,0.0000
P00025=3.643,0.007,-2.585,0.0000,0.0000,0.0000
P00026=2.644,0.055,-2.583,0.0000,0.0000,0.0000
P00027=2.278,0.099,-4.210,0.0000,0.0000,0.0000
P00028=-1.778,-0.182,-2.050,0.0000,0.0000,0.0000
P00029=1.749,4.006,-0.261,0.0000,0.0000,0.0000
P00030=-0.014,-0.768,0.131,0.0000,0.0000,0.0000
P00031=-0.170,0.039,-0.647,0.0000,0.0000,0.0000
P00032=-0.423,0.157,3.222,0.0000,0.0000,0.0000
P00033=0.854,-1.099,3.047,0.0000,0.0000,0.0000
///RCONF 0,0,0,0,1,0,0,0,0,0,0,0,0,0,0,0,0,0,0,0,0,0,0,0
P00034=-8.151,9.743,-4.393,0.0000,0.0000,0.0000
///RCONF 0,0,0,0,0,0,0,0,0,0,0,0,0,0,0,0,0,0,0,0,0,0,0,0
P00035=0.390,-0.027,1.040,0.0000,0.0000,0.0000
P00036=-2.434,0.084,0.197,0.0000,0.0000,0.0000
P00037=-1.075,5.090,-3.949,0.0000,0.0000,0.0000
P00038=0.174,-1.527,-10.860,0.0000,0.0000,0.0000
P00039=-0.109,1.838,-0.266,0.0000,0.0000,0.0000
P00040=2.716,-0.016,3.014,0.0000,0.0000,0.0000
//INST
///DATE 2024/12/09 21:51
///ATTR SC,RW
///GROUP1 RB1,BS1
///GROUP2 ST1
NOP
'X2_51(P)(-165,-90)
MOVJ C00000 BC00000 VJ=100.00  +MOVJ EC00000 VJ=100.00
MOVJ C00001 BC00001 VJ=100.00  +MOVJ EC00001 VJ=100.00
MOVJ C00002 BC00002 VJ=100.00  +MOVJ EC00002 VJ=100.00
'Path S3231
SFTOF3D
MOVJ C00003 BC00003 VJ=100.00  +MOVJ EC00003 VJ=100.00
MOVL C00004 BC00004 V=800.0  +MOVJ EC00004 VJ=100.00
SMOVL C00005 BC00005 V=166.7  +MOVJ EC00005
SREFP 3 C00006 BC00006  +REFP EC00006
CALL JOB:SEARCH-R1-S13D
SET P021 P006
SFTON3D P021
SMOVL C00007 BC00007 V=166.7  +MOVJ EC00007
SREFP 3 C00008 BC00008  +REFP EC00008
CALL JOB:SEARCH-R1-S13D
SET P021 P006
SFTON3D P021
SMOVL C00009 BC00009 V=166.7  +MOVJ EC00009
MOVL C00010 BC00010 V=1000.0  +MOVJ EC00010 VJ=100.00
'EndPath S3231
MOVJ C00011 BC00011 VJ=100.00  +MOVJ EC00011 VJ=100.00
'Path S3232
SFTOF3D
MOVJ C00012 BC00012 VJ=100.00  +MOVJ EC00012 VJ=100.00
MOVL C00013 BC00013 V=800.0  +MOVJ EC00013 VJ=100.00
SMOVL C00014 BC00014 V=166.7  +MOVJ EC00014
SREFP 3 C00015 BC00015  +REFP EC00015
CALL JOB:SEARCH-R1-S13D
SET P022 P006
SFTON3D P022
SMOVL C00016 BC00016 V=166.7  +MOVJ EC00016
SREFP 3 C00017 BC00017  +REFP EC00017
CALL JOB:SEARCH-R1-S13D
SET P022 P006
SFTON3D P022
SMOVL C00018 BC00018 V=166.7  +MOVJ EC00018
MOVL C00019 BC00019 V=1000.0  +MOVJ EC00019 VJ=100.00
'EndPath S3232
MOVJ C00020 BC00020 VJ=100.00  +MOVJ EC00020 VJ=100.00
'Path S3233
SFTOF3D
MOVJ C00021 BC00021 VJ=100.00  +MOVJ EC00021 VJ=100.00
MOVL C00022 BC00022 V=800.0  +MOVJ EC00022 VJ=100.00
SMOVL C00023 BC00023 V=166.7  +MOVJ EC00023
SREFP 3 C00024 BC00024  +REFP EC00024
CALL JOB:SEARCH-R1-S13D
SET P023 P006
SFTON3D P023
SMOVL C00025 BC00025 V=166.7  +MOVJ EC00025
SREFP 3 C00026 BC00026  +REFP EC00026
CALL JOB:SEARCH-R1-S13D
SET P023 P006
SFTON3D P023
SMOVL C00027 BC00027 V=166.7  +MOVJ EC00027
MOVL C00028 BC00028 V=1000.0  +MOVJ EC00028 VJ=100.00
'EndPath S3233
MOVJ C00029 BC00029 VJ=100.00  +MOVJ EC00029 VJ=100.00
'Path S3234
SFTOF3D
MOVJ C00030 BC00030 VJ=100.00  +MOVJ EC00030 VJ=100.00
MOVL C00031 BC00031 V=800.0  +MOVJ EC00031 VJ=100.00
SMOVL C00032 BC00032 V=166.7  +MOVJ EC00032
SREFP 3 C00033 BC00033  +REFP EC00033
CALL JOB:SEARCH-R1-S13D
SET P024 P006
SFTON3D P024
SMOVL C00034 BC00034 V=166.7  +MOVJ EC00034
SREFP 3 C00035 BC00035  +REFP EC00035
CALL JOB:SEARCH-R1-S13D
SET P024 P006
SFTON3D P024
SMOVL C00036 BC00036 V=166.7  +MOVJ EC00036
MOVL C00037 BC00037 V=1000.0  +MOVJ EC00037 VJ=100.00
'EndPath S3234
MOVJ C00038 BC00038 VJ=100.00  +MOVJ EC00038 VJ=100.00
'Path S3235
SFTOF3D
MOVJ C00039 BC00039 VJ=100.00  +MOVJ EC00039 VJ=100.00
MOVL C00040 BC00040 V=800.0  +MOVJ EC00040 VJ=100.00
SMOVL C00041 BC00041 V=166.7  +MOVJ EC00041
SREFP 3 C00042 BC00042  +REFP EC00042
CALL JOB:SEARCH-R1-S13D
SET P025 P006
SFTON3D P025
SMOVL C00043 BC00043 V=166.7  +MOVJ EC00043
SREFP 3 C00044 BC00044  +REFP EC00044
CALL JOB:SEARCH-R1-S13D
SET P025 P006
SFTON3D P025
SMOVL C00045 BC00045 V=166.7  +MOVJ EC00045
MOVL C00046 BC00046 V=1000.0  +MOVJ EC00046 VJ=100.00
'EndPath S3235
MOVJ C00047 BC00047 VJ=100.00  +MOVJ EC00047 VJ=100.00
'Path S3236
SFTOF3D
MOVJ C00048 BC00048 VJ=100.00  +MOVJ EC00048 VJ=100.00
MOVL C00049 BC00049 V=800.0  +MOVJ EC00049 VJ=100.00
SMOVL C00050 BC00050 V=166.7  +MOVJ EC00050
SREFP 3 C00051 BC00051  +REFP EC00051
CALL JOB:SEARCH-R1-S13D
SET P026 P006
SFTON3D P026
SMOVL C00052 BC00052 V=166.7  +MOVJ EC00052
SREFP 3 C00053 BC00053  +REFP EC00053
CALL JOB:SEARCH-R1-S13D
SET P026 P006
SFTON3D P026
SMOVL C00054 BC00054 V=166.7  +MOVJ EC00054
MOVL C00055 BC00055 V=800.0  +MOVJ EC00055 VJ=100.00
MOVL C00056 BC00056 V=1000.0  +MOVJ EC00056 VJ=100.00
'EndPath S3236
'obrot
MOVJ C00057 BC00057 VJ=100.00  +MOVJ EC00057 VJ=100.00
MOVJ C00058 BC00058 VJ=100.00  +MOVJ EC00058 VJ=100.00
MOVJ C00059 BC00059 VJ=100.00  +MOVJ EC00059 VJ=100.00
MOVJ C00060 BC00060 VJ=100.00  +MOVJ EC00060 VJ=100.00
MOVJ C00061 BC00061 VJ=100.00  +MOVJ EC00061 VJ=100.00
MOVJ C00062 BC00062 VJ=100.00  +MOVJ EC00062 VJ=100.00
'Path S3270
SFTOF3D
MOVJ C00063 BC00063 VJ=100.00  +MOVJ EC00063 VJ=100.00
MOVL C00064 BC00064 V=800.0  +MOVJ EC00064 VJ=100.00
SMOVL C00065 BC00065 V=166.7  +MOVJ EC00065
SREFP 3 C00066 BC00066  +REFP EC00066
CALL JOB:SEARCH-R1-S13D
SET P027 P006
SFTON3D P027
SMOVL C00067 BC00067 V=166.7  +MOVJ EC00067
SREFP 3 C00068 BC00068  +REFP EC00068
CALL JOB:SEARCH-R1-S13D
SET P027 P006
SFTON3D P027
SMOVL C00069 BC00069 V=166.7  +MOVJ EC00069
MOVL C00070 BC00070 V=800.0  +MOVJ EC00070 VJ=100.00
MOVL C00071 BC00071 V=1000.0  +MOVJ EC00071 VJ=100.00
'EndPath S3270
'Path S3271
SFTOF3D
MOVJ C00072 BC00072 VJ=100.00  +MOVJ EC00072 VJ=100.00
MOVL C00073 BC00073 V=800.0  +MOVJ EC00073 VJ=100.00
SMOVL C00074 BC00074 V=166.7  +MOVJ EC00074
SREFP 3 C00075 BC00075  +REFP EC00075
CALL JOB:SEARCH-R1-S13D
SET P028 P006
SFTON3D P028
SMOVL C00076 BC00076 V=166.7  +MOVJ EC00076
SREFP 3 C00077 BC00077  +REFP EC00077
CALL JOB:SEARCH-R1-S13D
SET P028 P006
SFTON3D P028
SMOVL C00078 BC00078 V=166.7  +MOVJ EC00078
MOVL C00079 BC00079 V=1000.0  +MOVJ EC00079 VJ=100.00
'EndPath S3271
MOVJ C00080 BC00080 VJ=100.00  +MOVJ EC00080 VJ=100.00
'Path S3271
SFTOF3D
MOVJ C00081 BC00081 VJ=100.00  +MOVJ EC00081 VJ=100.00
MOVL C00082 BC00082 V=800.0  +MOVJ EC00082 VJ=100.00
SMOVL C00083 BC00083 V=166.7  +MOVJ EC00083
SREFP 3 C00084 BC00084  +REFP EC00084
CALL JOB:SEARCH-R1-S13D
SET P029 P006
SFTON3D P029
SMOVL C00085 BC00085 V=166.7  +MOVJ EC00085
SREFP 3 C00086 BC00086  +REFP EC00086
CALL JOB:SEARCH-R1-S13D
SET P029 P006
SFTON3D P029
SMOVL C00087 BC00087 V=166.7  +MOVJ EC00087
MOVL C00088 BC00088 V=1000.0  +MOVJ EC00088 VJ=100.00
'EndPath S3271
'Path S3272
SFTOF3D
MOVJ C00089 BC00089 VJ=100.00  +MOVJ EC00089 VJ=100.00
MOVL C00090 BC00090 V=800.0  +MOVJ EC00090 VJ=100.00
SMOVL C00091 BC00091 V=166.7  +MOVJ EC00091
SREFP 3 C00092 BC00092  +REFP EC00092
CALL JOB:SEARCH-R1-S13D
SET P030 P006
SFTON3D P030
SMOVL C00093 BC00093 V=166.7  +MOVJ EC00093
SREFP 3 C00094 BC00094  +REFP EC00094
CALL JOB:SEARCH-R1-S13D
SET P030 P006
SFTON3D P030
SMOVL C00095 BC00095 V=166.7  +MOVJ EC00095
MOVL C00096 BC00096 V=1000.0  +MOVJ EC00096 VJ=100.00
'EndPath S3272
MOVJ C00097 BC00097 VJ=100.00  +MOVJ EC00097 VJ=100.00
MOVJ C00098 BC00098 VJ=100.00  +MOVJ EC00098 VJ=100.00
MOVJ C00099 BC00099 VJ=100.00  +MOVJ EC00099 VJ=100.00
'
MOVJ C00100 BC00100 VJ=100.00  +MOVJ EC00100 VJ=100.00
PAUSE
PAUSE
PAUSE
COMM MOVJ C00101 BC00101 VJ=100.00  +MOVJ EC00101 VJ=100.00
COMM MOVJ C00102 BC00102 VJ=100.00  +MOVJ EC00102 VJ=100.00
COMM MOVJ C00103 BC00103 VJ=100.00  +MOVJ EC00103 VJ=100.00
COMM MOVJ C00104 BC00104 VJ=100.00  +MOVJ EC00104 VJ=100.00
COMM MOVJ C00105 BC00105 VJ=100.00  +MOVJ EC00105 VJ=100.00
COMM 'Path S3272
COMM SFTOF3D
COMM MOVJ C00106 BC00106 VJ=100.00  +MOVJ EC00106 VJ=100.00
COMM MOVL C00107 BC00107 V=800.0  +MOVJ EC00107 VJ=100.00
COMM SMOVL C00108 BC00108 V=166.7  +MOVJ EC00108
COMM SREFP 3 C00109 BC00109  +REFP EC00109
COMM CALL JOB:SEARCH-R1-S13D
COMM SET P037 P006
COMM SFTON3D P037
COMM SMOVL C00110 BC00110 V=166.7  +MOVJ EC00110
COMM SREFP 3 C00111 BC00111  +REFP EC00111
COMM CALL JOB:SEARCH-R1-S13D
COMM SET P037 P006
COMM SFTON3D P037
COMM SMOVL C00112 BC00112 V=166.7  +MOVJ EC00112
COMM SMOVL C00113 BC00113 V=166.7  +MOVJ EC00113
COMM SREFP 3 C00114 BC00114  +REFP EC00114
COMM CALL JOB:SEARCH-R1-S13D
COMM SET P037 P006
COMM SFTON3D P037
COMM SMOVL C00115 BC00115 V=166.7  +MOVJ EC00115
COMM MOVL C00116 BC00116 V=1000.0  +MOVJ EC00116 VJ=100.00
COMM 'EndPath S3272
COMM 'Path S3273
COMM SFTOF3D
COMM MOVJ C00117 BC00117 VJ=100.00  +MOVJ EC00117 VJ=100.00
COMM MOVL C00118 BC00118 V=800.0  +MOVJ EC00118 VJ=100.00
COMM SMOVL C00119 BC00119 V=166.7  +MOVJ EC00119
COMM SREFP 3 C00120 BC00120  +REFP EC00120
COMM CALL JOB:SEARCH-R1-S13D
COMM SET P038 P006
COMM SFTON3D P038
COMM SMOVL C00121 BC00121 V=166.7  +MOVJ EC00121
COMM SREFP 3 C00122 BC00122  +REFP EC00122
COMM CALL JOB:SEARCH-R1-S13D
COMM SET P038 P006
COMM SFTON3D P038
COMM SMOVL C00123 BC00123 V=166.7  +MOVJ EC00123
COMM MOVL C00124 BC00124 V=1000.0  +MOVJ EC00124 VJ=100.00
COMM 'EndPath S3273
COMM MOVJ C00125 BC00125 VJ=100.00  +MOVJ EC00125 VJ=100.00
COMM 'Path S3273
COMM SFTOF3D
COMM MOVJ C00126 BC00126 VJ=100.00  +MOVJ EC00126 VJ=100.00
COMM MOVL C00127 BC00127 V=800.0  +MOVJ EC00127 VJ=100.00
COMM SMOVL C00128 BC00128 V=166.7  +MOVJ EC00128
COMM SREFP 3 C00129 BC00129  +REFP EC00129
COMM CALL JOB:SEARCH-R1-S13D
COMM SET P039 P006
COMM SFTON3D P039
COMM SMOVL C00130 BC00130 V=166.7  +MOVJ EC00130
COMM SREFP 3 C00131 BC00131  +REFP EC00131
COMM CALL JOB:SEARCH-R1-S13D
COMM SET P039 P006
COMM SFTON3D P039
COMM SMOVL C00132 BC00132 V=166.7  +MOVJ EC00132
COMM MOVL C00133 BC00133 V=1000.0  +MOVJ EC00133 VJ=100.00
COMM 'EndPath S3273
COMM 'Path S3274
COMM SFTOF3D
COMM MOVJ C00134 BC00134 VJ=100.00  +MOVJ EC00134 VJ=100.00
COMM MOVL C00135 BC00135 V=800.0  +MOVJ EC00135 VJ=100.00
COMM SMOVL C00136 BC00136 V=166.7  +MOVJ EC00136
COMM SREFP 3 C00137 BC00137  +REFP EC00137
COMM CALL JOB:SEARCH-R1-S13D
COMM SET P040 P006
COMM SFTON3D P040
COMM SMOVL C00138 BC00138 V=166.7  +MOVJ EC00138
COMM SREFP 3 C00139 BC00139  +REFP EC00139
COMM CALL JOB:SEARCH-R1-S13D
COMM SET P040 P006
COMM SFTON3D P040
COMM SMOVL C00140 BC00140 V=166.7  +MOVJ EC00140
COMM MOVL C00141 BC00141 V=1000.0  +MOVJ EC00141 VJ=100.00
COMM 'EndPath S3274
COMM MOVJ C00142 BC00142 VJ=100.00  +MOVJ EC00142 VJ=100.00
COMM MOVJ C00143 BC00143 VJ=100.00  +MOVJ EC00143 VJ=100.00
COMM MOVJ C00144 BC00144 VJ=100.00  +MOVJ EC00144 VJ=100.00
PAUSE
PAUSE
PAUSE
PAUSE
MOVJ C00145 BC00145 VJ=100.00  +MOVJ EC00145 VJ=100.00
MOVJ C00146 BC00146 VJ=100.00  +MOVJ EC00146 VJ=100.00
'
'Path S3274
SFTOF3D
MOVJ C00147 BC00147 VJ=100.00  +MOVJ EC00147 VJ=100.00
MOVL C00148 BC00148 V=800.0  +MOVJ EC00148 VJ=100.00
SMOVL C00149 BC00149 V=166.7  +MOVJ EC00149
SREFP 3 C00150 BC00150  +REFP EC00150
CALL JOB:SEARCH-R1-S13D
SET P034 P006
SFTON3D P034
SMOVL C00151 BC00151 V=166.7  +MOVJ EC00151
SREFP 3 C00152 BC00152  +REFP EC00152
CALL JOB:SEARCH-R1-S13D
SET P034 P006
SFTON3D P034
SMOVL C00153 BC00153 V=60.0  +MOVJ EC00153
MOVL C00154 BC00154 V=1000.0  +MOVJ EC00154 VJ=100.00
'EndPath S3274
'Path S3275
SFTOF3D
MOVJ C00155 BC00155 VJ=100.00  +MOVJ EC00155 VJ=100.00
MOVL C00156 BC00156 V=800.0  +MOVJ EC00156 VJ=100.00
SMOVL C00157 BC00157 V=166.7  +MOVJ EC00157
SREFP 3 C00158 BC00158  +REFP EC00158
CALL JOB:SEARCH-R1-S13D
SET P035 P006
SFTON3D P035
SMOVL C00159 BC00159 V=166.7  +MOVJ EC00159
SREFP 3 C00160 BC00160  +REFP EC00160
CALL JOB:SEARCH-R1-S13D
SET P035 P006
SFTON3D P035
SMOVL C00161 BC00161 V=166.7  +MOVJ EC00161
MOVL C00162 BC00162 V=1000.0  +MOVJ EC00162 VJ=100.00
'EndPath S3275
MOVJ C00163 BC00163 VJ=100.00  +MOVJ EC00163 VJ=100.00
'Path S3276
SFTOF3D
MOVJ C00164 BC00164 VJ=100.00  +MOVJ EC00164 VJ=100.00
MOVL C00165 BC00165 V=800.0  +MOVJ EC00165 VJ=100.00
SMOVL C00166 BC00166 V=166.7  +MOVJ EC00166
SREFP 3 C00167 BC00167  +REFP EC00167
CALL JOB:SEARCH-R1-S13D
SET P036 P006
SFTON3D P036
SMOVL C00168 BC00168 V=166.7  +MOVJ EC00168
SREFP 3 C00169 BC00169  +REFP EC00169
CALL JOB:SEARCH-R1-S13D
SET P036 P006
SFTON3D P036
SMOVL C00170 BC00170 V=166.7  +MOVJ EC00170
MOVL C00171 BC00171 V=1000.0  +MOVJ EC00171 VJ=100.00
'EndPath S3276
'Path S3277
SFTOF3D
MOVJ C00172 BC00172 VJ=100.00  +MOVJ EC00172 VJ=100.00
MOVL C00173 BC00173 V=800.0  +MOVJ EC00173 VJ=100.00
SMOVL C00174 BC00174 V=166.7  +MOVJ EC00174
SREFP 3 C00175 BC00175  +REFP EC00175
CALL JOB:SEARCH-R1-S13D
SET P031 P006
SFTON3D P031
SMOVL C00176 BC00176 V=166.7  +MOVJ EC00176
SREFP 3 C00177 BC00177  +REFP EC00177
CALL JOB:SEARCH-R1-S13D
SET P031 P006
SFTON3D P031
SMOVL C00178 BC00178 V=166.7  +MOVJ EC00178
MOVL C00179 BC00179 V=1000.0  +MOVJ EC00179 VJ=100.00
'EndPath S3277
MOVJ C00180 BC00180 VJ=100.00  +MOVJ EC00180 VJ=100.00
'Path S3278
SFTOF3D
MOVJ C00181 BC00181 VJ=100.00  +MOVJ EC00181 VJ=100.00
MOVL C00182 BC00182 V=800.0  +MOVJ EC00182 VJ=100.00
SMOVL C00183 BC00183 V=166.7  +MOVJ EC00183
SREFP 3 C00184 BC00184  +REFP EC00184
CALL JOB:SEARCH-R1-S13D
SET P032 P006
SFTON3D P032
SMOVL C00185 BC00185 V=166.7  +MOVJ EC00185
SREFP 3 C00186 BC00186  +REFP EC00186
CALL JOB:SEARCH-R1-S13D
SET P032 P006
SFTON3D P032
SMOVL C00187 BC00187 V=166.7  +MOVJ EC00187
MOVL C00188 BC00188 V=1000.0  +MOVJ EC00188 VJ=100.00
'EndPath S3278
'Path S3279
SFTOF3D
MOVJ C00189 BC00189 VJ=100.00  +MOVJ EC00189 VJ=100.00
MOVL C00190 BC00190 V=800.0  +MOVJ EC00190 VJ=100.00
SMOVL C00191 BC00191 V=166.7  +MOVJ EC00191
SREFP 3 C00192 BC00192  +REFP EC00192
CALL JOB:SEARCH-R1-S13D
SET P033 P006
SFTON3D P033
SMOVL C00193 BC00193 V=166.7  +MOVJ EC00193
SREFP 3 C00194 BC00194  +REFP EC00194
CALL JOB:SEARCH-R1-S13D
SET P033 P006
SFTON3D P033
SMOVL C00195 BC00195 V=166.7  +MOVJ EC00195
MOVL C00196 BC00196 V=1000.0  +MOVJ EC00196 VJ=100.00
'EndPath S3279
'
MOVJ C00197 BC00197 VJ=100.00  +MOVJ EC00197 VJ=100.00
MOVJ C00198 BC00198 VJ=100.00  +MOVJ EC00198 VJ=100.00
'
'
'Path W3280
SFTOF3D
SFTON3D P034
MOVJ C00199 BC00199 VJ=100.00  +MOVJ EC00199 VJ=100.00
SMOVL C00200 BC00200 V=800.0  +MOVJ EC00200
SMOVL C00201 BC00201 V=166.7 PL=0  +MOVJ EC00201
MACRO1 MJ#(0) ARGF21
ARCON
SMOVL C00202 BC00202 V=11.7  +MOVJ EC00202
ARCOF
SMOVL C00203 BC00203 V=800.0  +MOVJ EC00203
SMOVL C00204 BC00204 V=1000.0  +MOVJ EC00204
SFTOF3D
'EndPath W3280
'Path W3281
SFTOF3D
SFTON3D P035
MOVJ C00205 BC00205 VJ=100.00  +MOVJ EC00205 VJ=100.00
SMOVL C00206 BC00206 V=800.0  +MOVJ EC00206
SMOVL C00207 BC00207 V=166.7 PL=0  +MOVJ EC00207
ARCON
SMOVL C00208 BC00208 V=11.7  +MOVJ EC00208
ARCOF
SMOVL C00209 BC00209 V=800.0  +MOVJ EC00209
SMOVL C00210 BC00210 V=1000.0  +MOVJ EC00210
SFTOF3D
'EndPath W3281
MOVJ C00211 BC00211 VJ=100.00  +MOVJ EC00211 VJ=100.00
'Path W3282
SFTOF3D
SFTON3D P036
MOVJ C00212 BC00212 VJ=100.00  +MOVJ EC00212 VJ=100.00
SMOVL C00213 BC00213 V=800.0  +MOVJ EC00213
SMOVL C00214 BC00214 V=166.7 PL=0  +MOVJ EC00214
ARCON
SMOVL C00215 BC00215 V=11.7  +MOVJ EC00215
ARCOF
SMOVL C00216 BC00216 V=800.0  +MOVJ EC00216
SMOVL C00217 BC00217 V=1000.0  +MOVJ EC00217
SFTOF3D
'EndPath W3282
'Path W3283
SFTOF3D
SFTON3D P031
MOVJ C00218 BC00218 VJ=100.00  +MOVJ EC00218 VJ=100.00
SMOVL C00219 BC00219 V=800.0  +MOVJ EC00219
SMOVL C00220 BC00220 V=166.7 PL=0  +MOVJ EC00220
ARCON
SMOVL C00221 BC00221 V=11.7  +MOVJ EC00221
ARCOF
SMOVL C00222 BC00222 V=800.0  +MOVJ EC00222
SMOVL C00223 BC00223 V=1000.0  +MOVJ EC00223
SFTOF3D
'EndPath W3283
MOVJ C00224 BC00224 VJ=100.00  +MOVJ EC00224 VJ=100.00
'Path W3284
SFTOF3D
SFTON3D P032
MOVJ C00225 BC00225 VJ=100.00  +MOVJ EC00225 VJ=100.00
SMOVL C00226 BC00226 V=800.0  +MOVJ EC00226
SMOVL C00227 BC00227 V=166.7 PL=0  +MOVJ EC00227
ARCON
SMOVL C00228 BC00228 V=11.7  +MOVJ EC00228
ARCOF
SMOVL C00229 BC00229 V=800.0  +MOVJ EC00229
SMOVL C00230 BC00230 V=1000.0  +MOVJ EC00230
SFTOF3D
'EndPath W3284
'Path W3285
SFTOF3D
SFTON3D P033
MOVJ C00231 BC00231 VJ=100.00  +MOVJ EC00231 VJ=100.00
SMOVL C00232 BC00232 V=800.0  +MOVJ EC00232
SMOVL C00233 BC00233 V=166.7 PL=0  +MOVJ EC00233
ARCON
SMOVL C00234 BC00234 V=11.7  +MOVJ EC00234
ARCOF
SMOVL C00235 BC00235 V=800.0  +MOVJ EC00235
SMOVL C00236 BC00236 V=1000.0  +MOVJ EC00236
SFTOF3D
'EndPath W3285
'obrot
MOVJ C00237 BC00237 VJ=100.00  +MOVJ EC00237 VJ=100.00
MOVJ C00238 BC00238 VJ=100.00  +MOVJ EC00238 VJ=100.00
COMM MOVJ C00239 BC00239 VJ=100.00  +MOVJ EC00239 VJ=100.00
COMM MOVJ C00240 BC00240 VJ=100.00  +MOVJ EC00240 VJ=100.00
COMM MOVJ C00241 BC00241 VJ=100.00  +MOVJ EC00241 VJ=100.00
COMM 'Path W3267
COMM SFTOF3D
COMM SFTON3D P040
COMM MOVJ C00242 BC00242 VJ=100.00  +MOVJ EC00242 VJ=100.00
COMM SMOVL C00243 BC00243 V=800.0  +MOVJ EC00243
COMM SMOVL C00244 BC00244 V=166.7 PL=0  +MOVJ EC00244
COMM MACRO1 MJ#(0) ARGF9
COMM ARCON
COMM SFTON3D P039
COMM SMOVL C00245 BC00245 V=10.0  +MOVJ EC00245
COMM ARCOF
COMM SMOVL C00246 BC00246 V=800.0  +MOVJ EC00246
COMM SMOVL C00247 BC00247 V=1000.0  +MOVJ EC00247
COMM SFTOF3D
COMM 'EndPath W3267
COMM MOVJ C00248 BC00248 VJ=100.00  +MOVJ EC00248 VJ=100.00
COMM 'Path W3269
COMM SFTOF3D
COMM SFTON3D P038
COMM MOVJ C00249 BC00249 VJ=100.00  +MOVJ EC00249 VJ=100.00
COMM SMOVL C00250 BC00250 V=800.0  +MOVJ EC00250
COMM SMOVL C00251 BC00251 V=150.0 PL=0  +MOVJ EC00251
COMM MACRO1 MJ#(0) ARGF21
COMM ARCON
COMM SMOVL C00252 BC00252 V=9.2  +MOVJ EC00252
COMM SFTON3D P037
COMM SMOVL C00253 BC00253 V=9.2  +MOVJ EC00253
COMM ARCOF
COMM SMOVL C00254 BC00254 V=800.0  +MOVJ EC00254
COMM SMOVL C00255 BC00255 V=1000.0  +MOVJ EC00255
COMM SFTOF3D
COMM 'EndPath W3269
COMM MOVJ C00256 BC00256 VJ=100.00  +MOVJ EC00256 VJ=100.00
COMM MOVJ C00257 BC00257 VJ=100.00  +MOVJ EC00257 VJ=100.00
COMM MOVJ C00258 BC00258 VJ=100.00  +MOVJ EC00258 VJ=100.00
COMM MOVJ C00259 BC00259 VJ=100.00  +MOVJ EC00259 VJ=100.00
COMM MOVJ C00260 BC00260 VJ=100.00  +MOVJ EC00260 VJ=100.00
MOVJ C00261 BC00261 VJ=100.00  +MOVJ EC00261 VJ=100.00
MOVJ C00262 BC00262 VJ=100.00  +MOVJ EC00262 VJ=100.00
MOVJ C00263 BC00263 VJ=100.00  +MOVJ EC00263 VJ=100.00
MOVJ C00264 BC00264 VJ=100.00  +MOVJ EC00264 VJ=100.00
'
'Path W3286
SFTOF3D
SFTON3D P021
MOVJ C00265 BC00265 VJ=100.00  +MOVJ EC00265 VJ=100.00
SMOVL C00266 BC00266 V=800.0  +MOVJ EC00266
SMOVL C00267 BC00267 V=166.7 PL=0  +MOVJ EC00267
ARCON
SMOVL C00268 BC00268 V=11.7  +MOVJ EC00268
ARCOF
SMOVL C00269 BC00269 V=800.0  +MOVJ EC00269
SMOVL C00270 BC00270 V=1000.0  +MOVJ EC00270
SFTOF3D
'EndPath W3286
MOVJ C00271 BC00271 VJ=100.00  +MOVJ EC00271 VJ=100.00
'Path W3287
SFTOF3D
SFTON3D P022
MOVJ C00272 BC00272 VJ=100.00  +MOVJ EC00272 VJ=100.00
SMOVL C00273 BC00273 V=800.0  +MOVJ EC00273
SMOVL C00274 BC00274 V=166.7 PL=0  +MOVJ EC00274
ARCON
SMOVL C00275 BC00275 V=11.7  +MOVJ EC00275
ARCOF
SMOVL C00276 BC00276 V=800.0  +MOVJ EC00276
SMOVL C00277 BC00277 V=1000.0  +MOVJ EC00277
SFTOF3D
'EndPath W3287
MOVJ C00278 BC00278 VJ=100.00  +MOVJ EC00278 VJ=100.00
'Path W3288
SFTOF3D
SFTON3D P023
MOVJ C00279 BC00279 VJ=100.00  +MOVJ EC00279 VJ=100.00
SMOVL C00280 BC00280 V=800.0  +MOVJ EC00280
SMOVL C00281 BC00281 V=166.7 PL=0  +MOVJ EC00281
ARCON
SMOVL C00282 BC00282 V=11.7  +MOVJ EC00282
ARCOF
SMOVL C00283 BC00283 V=800.0  +MOVJ EC00283
SMOVL C00284 BC00284 V=1000.0  +MOVJ EC00284
SFTOF3D
'EndPath W3288
MOVJ C00285 BC00285 VJ=100.00  +MOVJ EC00285 VJ=100.00
'Path W3289
SFTOF3D
SFTON3D P023
MOVJ C00286 BC00286 VJ=100.00  +MOVJ EC00286 VJ=100.00
SMOVL C00287 BC00287 V=800.0  +MOVJ EC00287
SMOVL C00288 BC00288 V=166.7 PL=0  +MOVJ EC00288
ARCON
SMOVL C00289 BC00289 V=11.7  +MOVJ EC00289
ARCOF
SMOVL C00290 BC00290 V=800.0  +MOVJ EC00290
SMOVL C00291 BC00291 V=1000.0  +MOVJ EC00291
SFTOF3D
'EndPath W3289
MOVJ C00292 BC00292 VJ=100.00  +MOVJ EC00292 VJ=100.00
'Path W3290
SFTOF3D
SFTON3D P022
MOVJ C00293 BC00293 VJ=100.00  +MOVJ EC00293 VJ=100.00
SMOVL C00294 BC00294 V=800.0  +MOVJ EC00294
SMOVL C00295 BC00295 V=166.7 PL=0  +MOVJ EC00295
ARCON
SMOVL C00296 BC00296 V=11.7  +MOVJ EC00296
ARCOF
SMOVL C00297 BC00297 V=800.0  +MOVJ EC00297
SMOVL C00298 BC00298 V=1000.0  +MOVJ EC00298
SFTOF3D
'EndPath W3290
MOVJ C00299 BC00299 VJ=100.00  +MOVJ EC00299 VJ=100.00
'Path W3291
SFTOF3D
SFTON3D P021
MOVJ C00300 BC00300 VJ=100.00  +MOVJ EC00300 VJ=100.00
SMOVL C00301 BC00301 V=800.0  +MOVJ EC00301
SMOVL C00302 BC00302 V=166.7 PL=0  +MOVJ EC00302
ARCON
SMOVL C00303 BC00303 V=11.7  +MOVJ EC00303
ARCOF
SMOVL C00304 BC00304 V=800.0  +MOVJ EC00304
SMOVL C00305 BC00305 V=1000.0  +MOVJ EC00305
SFTOF3D
'EndPath W3291
MOVJ C00306 BC00306 VJ=100.00  +MOVJ EC00306 VJ=100.00
MOVJ C00307 BC00307 VJ=100.00  +MOVJ EC00307 VJ=100.00
MOVJ C00308 BC00308 VJ=100.00  +MOVJ EC00308 VJ=100.00
MOVJ C00309 BC00309 VJ=100.00  +MOVJ EC00309 VJ=100.00
'Path W3262
SFTOF3D
SFTON3D P028
MOVJ C00310 BC00310 VJ=100.00  +MOVJ EC00310 VJ=100.00
SMOVL C00311 BC00311 V=800.0  +MOVJ EC00311
SMOVL C00312 BC00312 V=166.7 PL=0  +MOVJ EC00312
ARCON
SFTON3D P027
SMOVL C00313 BC00313 V=9.2  +MOVJ EC00313
ARCOF
SMOVL C00314 BC00314 V=800.0  +MOVJ EC00314
SMOVL C00315 BC00315 V=1000.0  +MOVJ EC00315
SFTOF3D
'EndPath W3262
MOVJ C00316 BC00316 VJ=100.00  +MOVJ EC00316 VJ=100.00
'Path W3264
SFTOF3D
SFTON3D P030
MOVJ C00317 BC00317 VJ=100.00  +MOVJ EC00317 VJ=100.00
SMOVL C00318 BC00318 V=800.0  +MOVJ EC00318
SMOVL C00319 BC00319 V=166.7 PL=0  +MOVJ EC00319
MACRO1 MJ#(0) ARGF9
ARCON
SFTON3D P029
SMOVL C00320 BC00320 V=10.0  +MOVJ EC00320
ARCOF
SMOVL C00321 BC00321 V=800.0  +MOVJ EC00321
SMOVL C00322 BC00322 V=1000.0  +MOVJ EC00322
SFTOF3D
'EndPath W3264
MOVJ C00323 BC00323 VJ=100.00  +MOVJ EC00323 VJ=100.00
MOVJ C00324 BC00324 VJ=30.00  +MOVJ EC00324 VJ=30.00
MOVJ C00325 BC00325 VJ=30.00  +MOVJ EC00325 VJ=30.00
MOVJ C00326 BC00326 VJ=30.00  +MOVJ EC00326 VJ=30.00
SFTON3D P027
SMOVL C00327 BC00327 V=133.3  +MOVJ EC00327
ARCON
SMOVL C00328 BC00328 V=9.2  +MOVJ EC00328
ARCOF
SFTOF3D
SMOVL C00329 BC00329 V=166.7  +MOVJ EC00329
SMOVL C00330 BC00330 V=166.7  +MOVJ EC00330
SFTON3D P029
SMOVL C00331 BC00331 V=166.7  +MOVJ EC00331
ARCON
SMOVL C00332 BC00332 V=10.0  +MOVJ EC00332
ARCOF
SFTOF3D
SMOVL C00333 BC00333 V=250.0  +MOVJ EC00333
SMOVL C00334 BC00334 V=250.0  +MOVJ EC00334
MOVJ C00335 BC00335 VJ=30.00  +MOVJ EC00335 VJ=30.00
MOVJ C00336 BC00336 VJ=100.00  +MOVJ EC00336 VJ=100.00
END
